{attribute 'GeneratedUsingTerminal: ELX3204-0000-0016'}
{attribute addProperty BoxType "ELX3204-0000-0016"}
{attribute addProperty Id "RTD_Inputs_Channel_1AT %I*RTD_Inputs_Channel_4A3944819RTD_Inputs_Channel_2AT %I*RTD_Inputs_Channel_4A3944819RTD_Inputs_Channel_3AT %I*RTD_Inputs_Channel_4A3944819RTD_Inputs_Channel_4AT %I*RTD_Inputs_Channel_4A3944819WcStateAT %I*WcState_9091E0EB2InfoDataAT %I*InfoData_94A18F5E2"}
{attribute addProperty CRC "3548533592"}
{attribute addProperty Size "40"}
TYPE ELX3204_D3825358 EXTENDS EtcSlaveTerminalBase_947E5A46 :
STRUCT
	{attribute addProperty Name "RTD_Inputs_Channel_1"}
	RTD_Inputs_Channel_1 : RTD_Inputs_Channel_4A394481;
	{attribute addProperty Name "RTD_Inputs_Channel_2"}
	RTD_Inputs_Channel_2 : RTD_Inputs_Channel_4A394481;
	{attribute addProperty Name "RTD_Inputs_Channel_3"}
	RTD_Inputs_Channel_3 : RTD_Inputs_Channel_4A394481;
	{attribute addProperty Name "RTD_Inputs_Channel_4"}
	RTD_Inputs_Channel_4 : RTD_Inputs_Channel_4A394481;
	{attribute addProperty Name "WcState"}
	WcState : WcState_9091E0EB;
	{attribute addProperty Name "InfoData"}
	InfoData : InfoData_94A18F5E;
END_STRUCT
END_TYPE

(* stored: Version 1.2.0.0, ProductVersion 3.1.4024.9
   DUT ELX3204_D3825358: Id {a68fed23-bd53-4dae-a4ac-0a8bdbc876b7} *)
